TYPE ST175_Recipe_t :
STRUCT
    isTypeSmartOrMini : BOOL; // do we need to run the laser twice on the same mover?
    file_name         : STRING;
END_STRUCT
END_TYPE

(* stored: Version 1.1.0.1, ProductVersion 3.1.4024.6
   DUT ST175_Recipe_t: Id {4e48d2da-cc5e-43a6-bc3e-2f0f9b670724} *)
